{attribute 'qualified_only'}
{attribute 'strict'}
TYPE Movement :
(
	ON := 1,
	OFF := 0
);
END_TYPE

(* stored: Version 1.1.0.1, ProductVersion 3.1.4024.13
   EnumerationTextList Movement: Id {4720dce9-a4c0-4815-825e-89d51033f37d} *)
